PROGRAM PRG_PLAS_03_PackToStackerCtrl
VAR
	bShiftStackerDataSet						: BOOL;

	fbMovePackToStacker						: FB_T01_MovePackToStacker;
	fbFillInPackInfeedQueue					: FB_PLAS_MasterListFillInPack;

	aStackIndexDebug							: ARRAY[0..21] OF UDINT;

	fbDebugCNT								: FB_DEBUG_CounterArray;
	aCNTDebug							: ARRAY [1..10] OF UDINT;
	bResetCNT							: BOOL;

END_VAR
VAR // added by the converter: edge detectors and wires of the graphical bodies
    _w1, _w2 : BOOL;
END_VAR

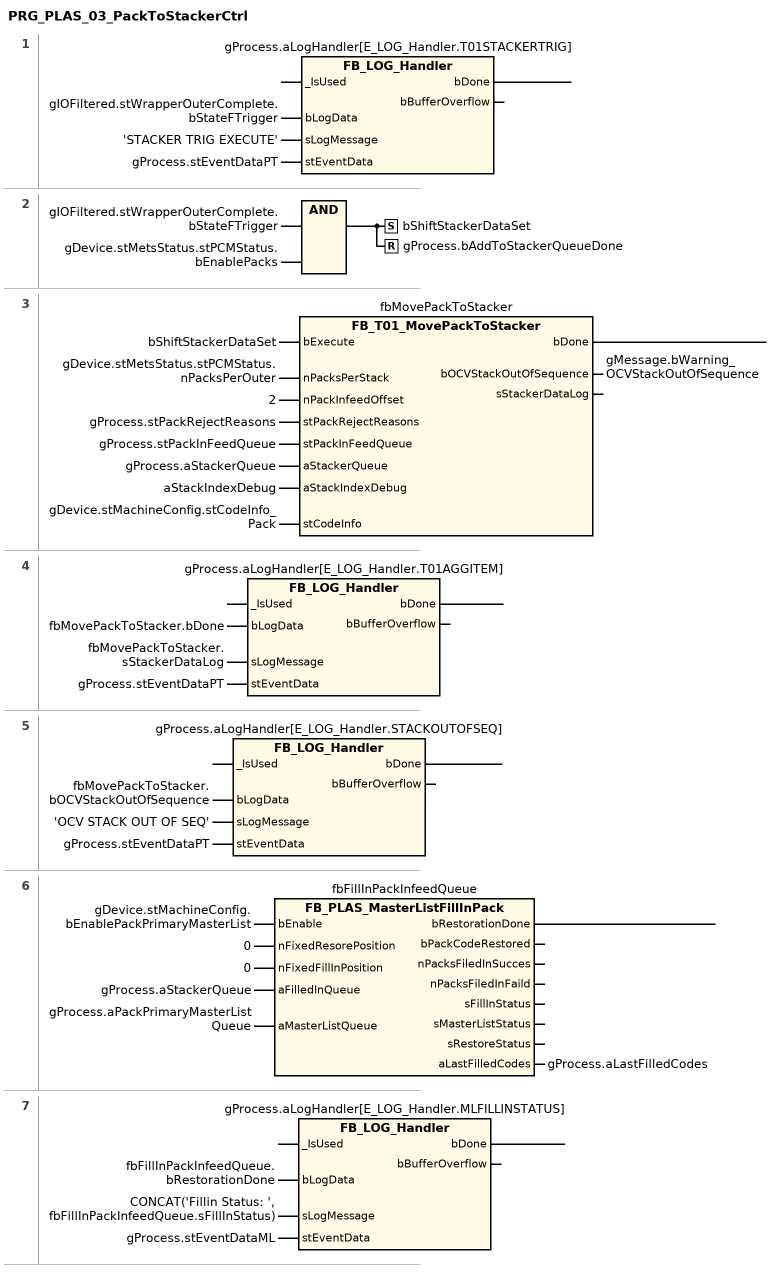
// NETWORK 1
gProcess.aLogHandler[E_LOG_Handler.T01STACKERTRIG](
    bLogData := gIOFiltered.stWrapperOuterComplete.bStateFTrigger,
    sLogMessage := 'STACKER TRIG EXECUTE',
    stEventData := gProcess.stEventDataPT); // FB_LOG_Handler

// NETWORK 2
_w1 := gIOFiltered.stWrapperOuterComplete.bStateFTrigger AND gDevice.stMetsStatus.stPCMStatus.bEnablePacks;
bShiftStackerDataSet S= _w1;
gProcess.bAddToStackerQueueDone R= _w1;

// NETWORK 3
fbMovePackToStacker(
    bExecute := bShiftStackerDataSet,
    nPacksPerStack := gDevice.stMetsStatus.stPCMStatus.nPacksPerOuter,
    nPackInfeedOffset := 2,
    stPackRejectReasons := gProcess.stPackRejectReasons,
    stPackInFeedQueue := gProcess.stPackInFeedQueue,
    aStackerQueue := gProcess.aStackerQueue,
    aStackIndexDebug := aStackIndexDebug,
    stCodeInfo := gDevice.stMachineConfig.stCodeInfo_Pack,
    bOCVStackOutOfSequence => gMessage.bWarning_OCVStackOutOfSequence); // FB_T01_MovePackToStacker

// NETWORK 4
gProcess.aLogHandler[E_LOG_Handler.T01AGGITEM](
    bLogData := fbMovePackToStacker.bDone,
    sLogMessage := fbMovePackToStacker.sStackerDataLog,
    stEventData := gProcess.stEventDataPT); // FB_LOG_Handler

// NETWORK 5
gProcess.aLogHandler[E_LOG_Handler.STACKOUTOFSEQ](
    bLogData := fbMovePackToStacker.bOCVStackOutOfSequence,
    sLogMessage := 'OCV STACK OUT OF SEQ',
    stEventData := gProcess.stEventDataPT); // FB_LOG_Handler

// NETWORK 6
fbFillInPackInfeedQueue(
    bEnable := gDevice.stMachineConfig.bEnablePackPrimaryMasterList,
    nFixedResorePosition := 0,
    nFixedFillInPosition := 0,
    aFilledInQueue := gProcess.aStackerQueue,
    aMasterListQueue := gProcess.aPackPrimaryMasterListQueue,
    aLastFilledCodes => gProcess.aLastFilledCodes); // FB_PLAS_MasterListFillInPack

// NETWORK 7
gProcess.aLogHandler[E_LOG_Handler.MLFILLINSTATUS](
    bLogData := fbFillInPackInfeedQueue.bRestorationDone,
    sLogMessage := CONCAT('Fillin Status: ', fbFillInPackInfeedQueue.sFillInStatus),
    stEventData := gProcess.stEventDataML); // FB_LOG_Handler

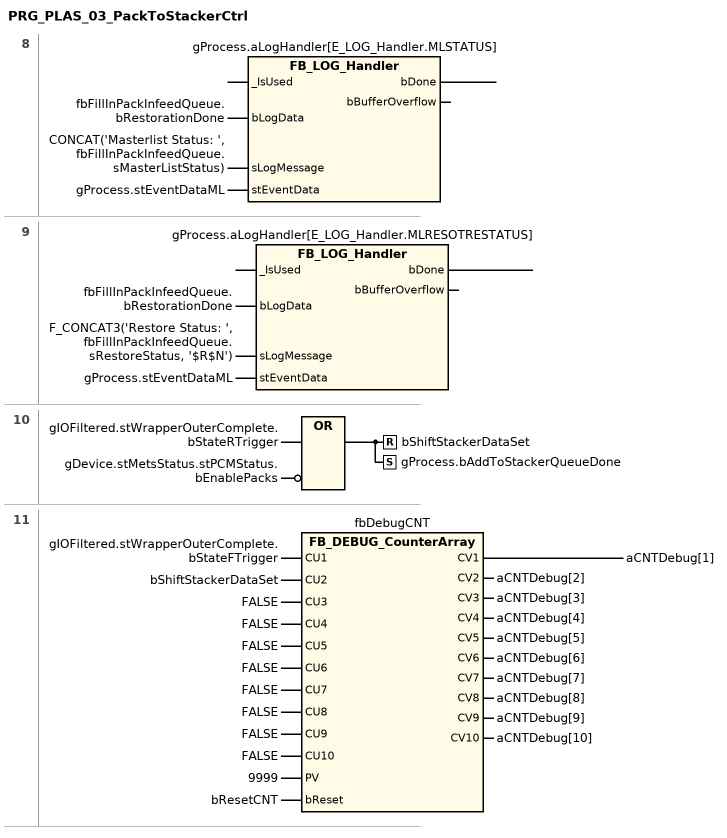
// NETWORK 8
gProcess.aLogHandler[E_LOG_Handler.MLSTATUS](
    bLogData := fbFillInPackInfeedQueue.bRestorationDone,
    sLogMessage := CONCAT('Masterlist Status: ',  fbFillInPackInfeedQueue.sMasterListStatus),
    stEventData := gProcess.stEventDataML); // FB_LOG_Handler

// NETWORK 9
gProcess.aLogHandler[E_LOG_Handler.MLRESOTRESTATUS](
    bLogData := fbFillInPackInfeedQueue.bRestorationDone,
    sLogMessage := F_CONCAT3('Restore Status: ',  fbFillInPackInfeedQueue.sRestoreStatus, '$R$N'),
    stEventData := gProcess.stEventDataML); // FB_LOG_Handler

// NETWORK 10
_w2 := gIOFiltered.stWrapperOuterComplete.bStateRTrigger OR NOT gDevice.stMetsStatus.stPCMStatus.bEnablePacks;
bShiftStackerDataSet R= _w2;
gProcess.bAddToStackerQueueDone S= _w2;

// NETWORK 11
fbDebugCNT(
    CU1 := gIOFiltered.stWrapperOuterComplete.bStateFTrigger,
    CU2 := bShiftStackerDataSet,
    CU3 := FALSE,
    CU4 := FALSE,
    CU5 := FALSE,
    CU6 := FALSE,
    CU7 := FALSE,
    CU8 := FALSE,
    CU9 := FALSE,
    CU10 := FALSE,
    PV := 9999,
    bReset := bResetCNT,
    CV2 => aCNTDebug[2],
    CV3 => aCNTDebug[3],
    CV4 => aCNTDebug[4],
    CV5 => aCNTDebug[5],
    CV6 => aCNTDebug[6],
    CV7 => aCNTDebug[7],
    CV8 => aCNTDebug[8],
    CV9 => aCNTDebug[9],
    CV10 => aCNTDebug[10]); // FB_DEBUG_CounterArray
aCNTDebug[1] := fbDebugCNT.CV1;

END_PROGRAM

(* stored: Version 1.1.0.1
   POU PRG_PLAS_03_PackToStackerCtrl: Id {9f899330-6bae-438d-ad6b-ff84a1331859}, SpecialFunc None *)
